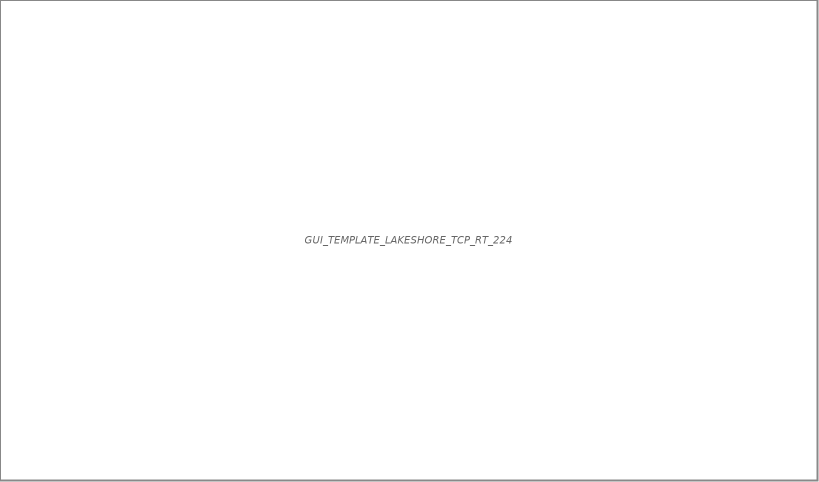
VISUALIZATION GUI_LAKESHORE_TCP_RT_224  // 819x482
    Frame (0,0 817x480)
        shows GUI_TEMPLATE_LAKESHORE_TCP_RT_224(m_Instance := MAIN.LS224_TCP_RT)
END_VISUALIZATION

(* stored: Version 1.1.0.1, ProductVersion 3.1.4022.16
   Visu GUI_LAKESHORE_TCP_RT_224: Id {52c696a1-dc09-41b8-980e-677f6dfd1a81} *)
